INTERFACE ITF_BaseComponent_HMI_Connector EXTENDS ITF_BaseComponent_HMI_Connector_View, ITF_BaseComponent_HMI_Connector_Command

END_INTERFACE

(* stored: Version 1.1.0.1
   Itf ITF_BaseComponent_HMI_Connector: Id {4a87bd4f-d701-0073-225c-a3573008b8a3} *)
